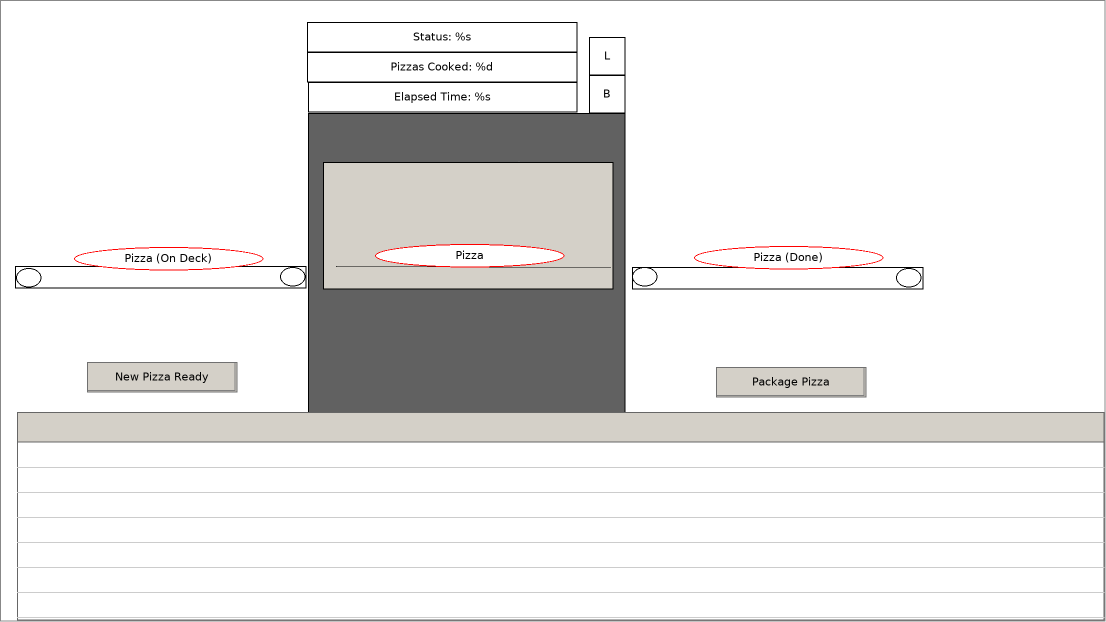
VISUALIZATION Visualization  // 1106x622
    Rectangle (308,113 317x477)
    Button (87,362 150x30), "New Pizza Ready"
        tap MAIN.bLoadPizza
    Button (716,367 150x30), "Package Pizza"
        tap MAIN.bRemovePizza
    Button (503,164 18x0)
    Rectangle (323,162 290x127)
    Rectangle (308,82 269x30), "Elapsed Time: %s", text variable: MAIN.fbMyPizzaOven.fbMyTimer.ET
    RoundedRectangle (15,266 291x22)
    RoundedRectangle (632,267 291x22)
    Ellipse (694,246 189x23), "Pizza (Done)", invisible if: NOT MAIN.fbMyPizzaOven.stPizzaDone.bExist
    Ellipse (74,247 189x23), "Pizza (On Deck)", invisible if: NOT MAIN.fbMyPizzaOven.stPizzaOnDeck.bExist
    Line (336,266) (610,267)
    Ellipse (375,244 189x23), "Pizza", invisible if: NOT MAIN.fbMyPizzaOven.stPizzaInOven.bExist
    RoundedRectangle (589,75 36x38), "B", colour toggle: MAIN.fbMyPizzaOven.bBuzzer
    RoundedRectangle (589,37 36x38), "L", colour toggle: MAIN.fbMyPizzaOven.bLight
    Rectangle (307,52 270x30), "Pizzas Cooked: %d", text variable: MAIN.fbMyPizzaOven.iTotalPizzasCooked
    Ellipse (16,268 25x19)
    Ellipse (280,267 25x19)
    Ellipse (632,267 25x19)
    Ellipse (896,268 25x19)
    Rectangle (307,22 270x30), "Status: %s", text variable: MAIN.fbMyPizzaOven.sStateDesc
    Table (17,412 1087x208), data array: HMI_VARS.arrPizzaHistory
        p3854506369: HMI_VARS.arrPizzaHistory[INDEX].bExist
        p1892666644: HMI_VARS.arrPizzaHistory[INDEX].dtTimeEnteredOven
        p338671338: HMI_VARS.arrPizzaHistory[INDEX].dtTimeExitedOven
        p2170511999: HMI_VARS.arrPizzaHistory[INDEX].tTimeInOven
        p3723444502: HMI_VARS.arrPizzaHistory[INDEX].eType
END_VISUALIZATION

(* stored: Version 1.1.0.1, ProductVersion 3.1.0.26
   Visu Visualization: Id {67ce955f-c384-417c-86be-b3381fccb77a} *)
